INTERFACE I_Position EXTENDS __SYSTEM.IQueryInterface

PROPERTY CurrentPosition : LREAL
GET
END_GET
END_PROPERTY

PROPERTY IsStationary : bool
GET
END_GET
END_PROPERTY

METHOD MoveByDistance : HRESULT
VAR_INPUT
	Distance : MC_LREAL;
	Velocity : MC_LREAL;
END_VAR
END_METHOD

METHOD MoveToModuloPosition : HRESULT
VAR_INPUT
	Position : MC_LREAL;
	Velocity : MC_LREAL;
END_VAR
END_METHOD

METHOD MoveToPosition : HRESULT
VAR_INPUT
	Position : MC_LREAL;
	Velocity : MC_LREAL;
END_VAR
END_METHOD

END_INTERFACE

(* stored: Version 1.1.0.1
   Itf I_Position: Id {67ee2d44-07ee-4a7f-8cf0-2ba796d7942a}
   Property CurrentPosition: Id {205db87f-f7bb-4e74-ad59-4c514b54dda0}
   Get Get: Id {27e51b78-62c8-44b7-a5f2-0d1b26ebf193}
   Property IsStationary: Id {27d390c2-fbca-4a5c-bcc1-15c4bbbbfc4f}
   Get Get: Id {e895ea74-610a-464d-8612-26e8bb00b426}
   Method MoveByDistance: Id {a5b81455-a8f6-4114-80eb-0d55f77596a7}
   Method MoveToModuloPosition: Id {41ccc185-4245-4d0a-9e77-77dc1b4d301f}
   Method MoveToPosition: Id {c5eac34c-4010-4d8b-8622-96313c7f08cf} *)
